# EPICS autosave request: mcaApp/Db/DSA2000_HVPS_settings.req
# FILE... icb_hvps_settings.req
# USAGE.. icb_hvps.db fields autosave'd.
$(P)$(HVPS)VOLTS
$(P)$(HVPS)RANGE
$(P)$(HVPS)INHIBIT_LEVEL
$(P)$(HVPS)READBACK_SCAN.SCAN
